// Mitsubishi GX Works2 project: PROJETO-ATUALIZADO   PLC: Q03UDV

PROGRAM MAIN
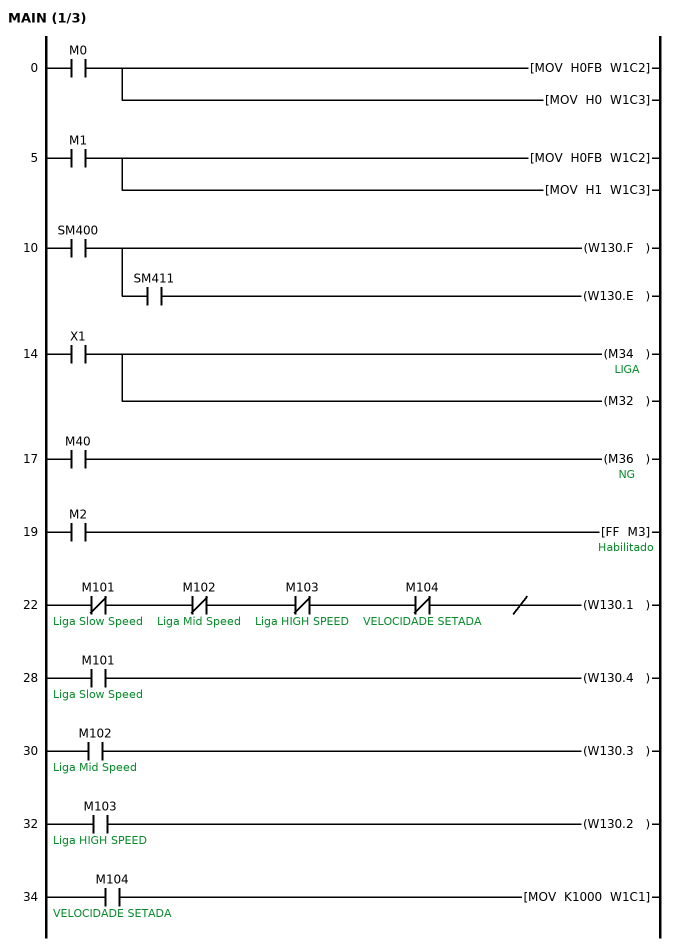
0     LD      M0
      MOV     H0FB W1C2
      MOV     H0 W1C3
5     LD      M1
      MOV     H0FB W1C2
      MOV     H1 W1C3
10    LD      SM400
      OUT     W130.F
      AND     SM411
      OUT     W130.E
14    LD      X1
      OUT     M34  ; LIGA
      OUT     M32
17    LD      M40
      OUT     M36  ; NG
19    LD      M2
      FF      M3  ; Habilitado
22    LDI     M101  ; Liga Slow Speed
      ANI     M102  ; Liga Mid Speed
      ANI     M103  ; Liga HIGH SPEED
      ANI     M104  ; VELOCIDADE SETADA
      INV
      OUT     W130.1
28    LD      M101  ; Liga Slow Speed
      OUT     W130.4
30    LD      M102  ; Liga Mid Speed
      OUT     W130.3
32    LD      M103  ; Liga HIGH SPEED
      OUT     W130.2
34    LD      M104  ; VELOCIDADE SETADA
      MOV     K1000 W1C1
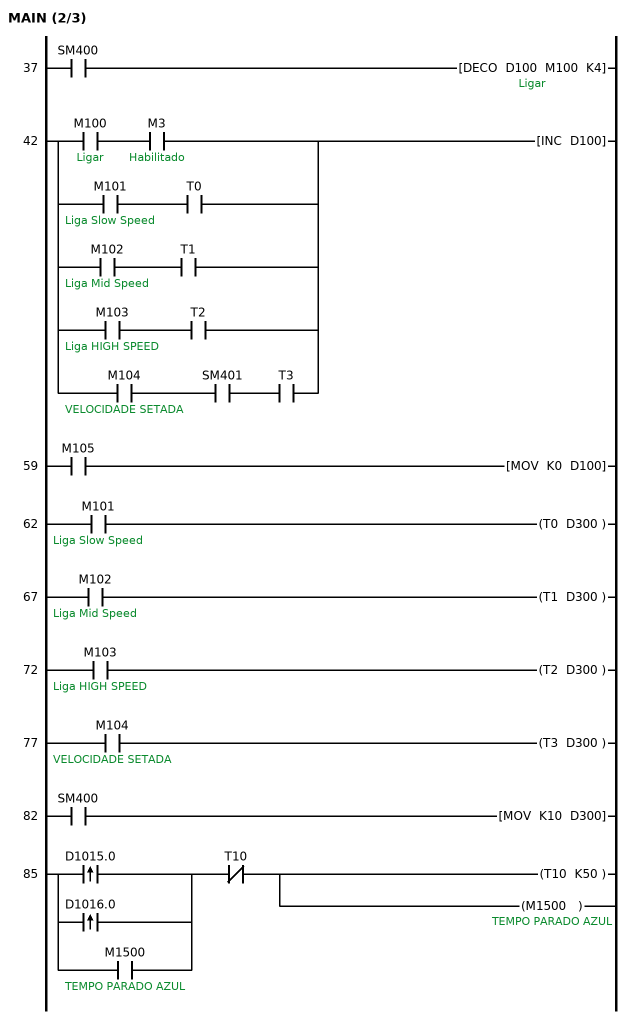
37    LD      SM400
      DECO    D100 M100 K4  ; Ligar
42    LD      M100  ; Ligar
      AND     M3  ; Habilitado
      LD      M101  ; Liga Slow Speed
      AND     T0
      ORB
      LD      M102  ; Liga Mid Speed
      AND     T1
      ORB
      LD      M103  ; Liga HIGH SPEED
      AND     T2
      ORB
      LD      M104  ; VELOCIDADE SETADA
      AND     SM401
      AND     T3
      ORB
      INC     D100
59    LD      M105
      MOV     K0 D100
62    LD      M101  ; Liga Slow Speed
      OUT     T0 D300
67    LD      M102  ; Liga Mid Speed
      OUT     T1 D300
72    LD      M103  ; Liga HIGH SPEED
      OUT     T2 D300
77    LD      M104  ; VELOCIDADE SETADA
      OUT     T3 D300
82    LD      SM400
      MOV     K10 D300
85    LDP     D1015.0
      ORP     D1016.0
      OR      M1500  ; TEMPO PARADO AZUL
      ANI     T10
      OUT     T10 K50
      OUT     M1500  ; TEMPO PARADO AZUL
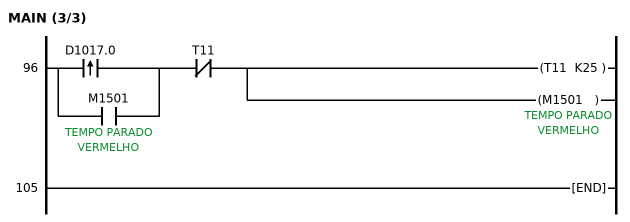
96    LDP     D1017.0
      OR      M1501  ; TEMPO PARADO VERMELHO
      ANI     T11
      OUT     T11 K25
      OUT     M1501  ; TEMPO PARADO VERMELHO
105   END
END_PROGRAM

// device comments not shown above
M250  ; LIGA
M1000  ; LIGA
